Universal Robots PolyScope program: Square.urp

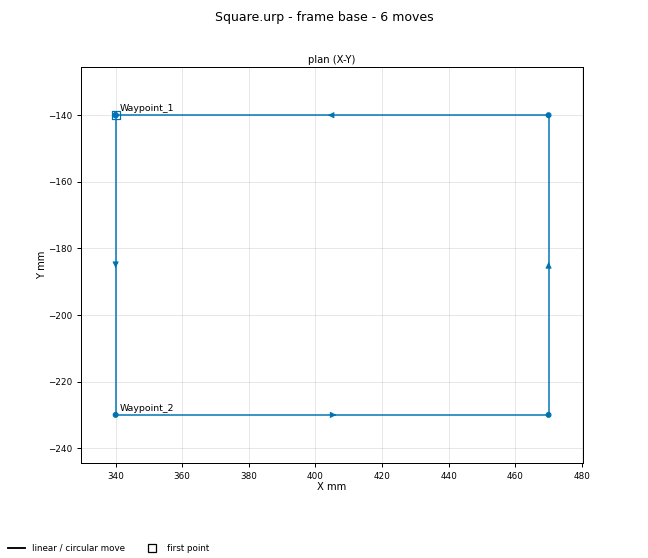
[picture p0: tool path of Square.urp in frame base, 6 of 6 moves have a stored position in this frame; points joined in program order, loops and branches not executed]
Program Square (installation=default directory=/programs createdIn=5.11.9.1010452 lastSavedIn=5.11.9.1010452 robotSerialNumber=20225200364)
Calibrated DH parameters: a=[0.00002, -0.569483, -0.54992, -0.00001, -0.000036, 0]; d=[0.180894, -146.691669, 192.918669, -46.053088, 0.119778, 0.115602]; alpha=[1.571425, -0.001534, 0.003359, 1.568739, -1.571477, 0]; deltaTheta=[0, 0.376258, -0.101074, -0.275185, -0.000002, 0]
Robot Program (runOnlyOnce=false)
  MoveL speed 250 mm/s, acceleration 1200 mm/s^2 (useActiveTCP=true) feature=Base
    Waypoint Waypoint_1: TCP in base x=340 y=-140 z=269 mm, rx=-0.2018 ry=3.135 rz=0 rad; joints [5.855, -66.957, -152.153, -50.845, 90.202, 88.508] deg; TCP offset x=0 y=0 z=0 mm, rx=0 ry=0 rz=0 rad
    Waypoint Waypoint_6: TCP in base x=340 y=-140 z=266.4 mm, rx=-0.2019 ry=3.135 rz=-0.0001 rad; joints [5.855, -67.287, -152.336, -50.334, 90.198, 88.509] deg; TCP offset x=0 y=0 z=0 mm, rx=0 ry=0 rz=0 rad
    Wait Sleep waitTime=0.5
    Waypoint Waypoint_2: TCP in base x=340 y=-230 z=267 mm, rx=-0.2018 ry=3.135 rz=0.0002 rad; joints [-9.021, -74.058, -148.67, -47.227, 90.197, 73.651] deg; TCP offset x=0 y=0 z=0 mm, rx=0 ry=0 rz=0 rad
    Waypoint Waypoint_3: TCP in base x=470 y=-230 z=267 mm, rx=-0.2019 ry=3.135 rz=0.0001 rad; joints [-6.693, -87.752, -138.202, -43.999, 90.169, 75.997] deg; TCP offset x=0 y=0 z=0 mm, rx=0 ry=0 rz=0 rad
    Waypoint Waypoint_4: TCP in base x=470 y=-140 z=266.8 mm, rx=-0.2018 ry=3.135 rz=0.0001 rad; joints [4.158, -84.239, -141.37, -44.343, 90.174, 86.848] deg; TCP offset x=0 y=0 z=0 mm, rx=0 ry=0 rz=0 rad
    Waypoint Waypoint_5: TCP in base x=340.004 y=-140 z=266.6 mm, rx=-0.2018 ry=3.135 rz=0 rad; joints [5.854, -67.262, -152.323, -50.367, 90.202, 88.509] deg; TCP offset x=0 y=0 z=0 mm, rx=0 ry=0 rz=0 rad
    Wait Sleep waitTime=1
